// Mitsubishi GX Developer project: 11-404八軸鎖螺絲機201107140830   PLC: FX1N

PROGRAM MAIN
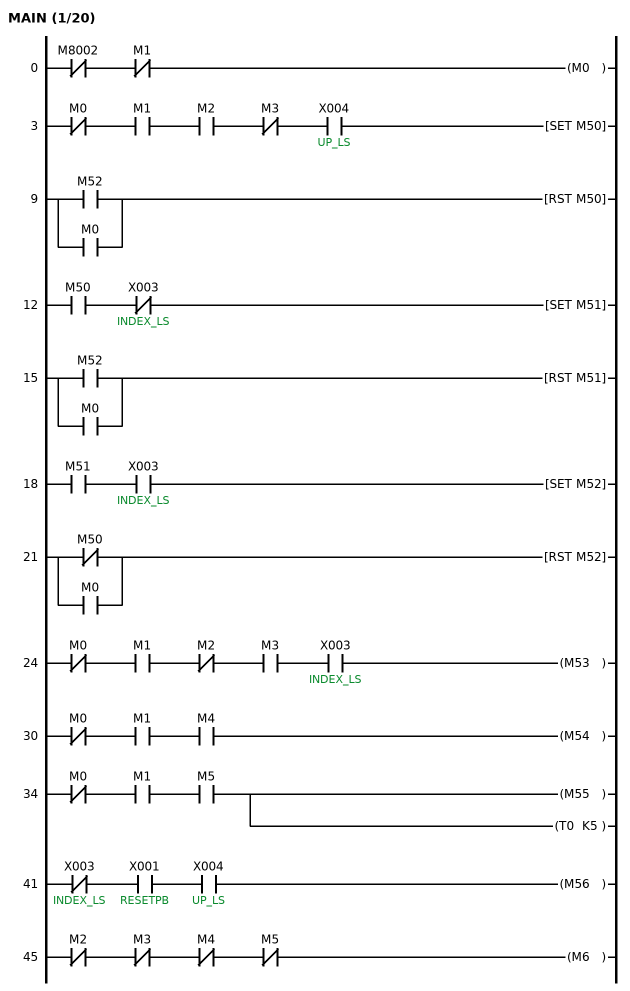
0     LDI     M8002
      ANI     M1
      OUT     M0
3     LDI     M0
      AND     M1
      AND     M2
      ANI     M3
      AND     X004  ; UP_LS
      SET     M50
9     LD      M52
      OR      M0
      RST     M50
12    LD      M50
      ANI     X003  ; INDEX_LS
      SET     M51
15    LD      M52
      OR      M0
      RST     M51
18    LD      M51
      AND     X003  ; INDEX_LS
      SET     M52
21    LDI     M50
      OR      M0
      RST     M52
24    LDI     M0
      AND     M1
      ANI     M2
      AND     M3
      AND     X003  ; INDEX_LS
      OUT     M53
30    LDI     M0
      AND     M1
      AND     M4
      OUT     M54
34    LDI     M0
      AND     M1
      AND     M5
      OUT     M55
      OUT     T0 K5
41    LDI     X003  ; INDEX_LS
      AND     X001  ; RESETPB
      AND     X004  ; UP_LS
      OUT     M56
45    LDI     M2
      ANI     M3
      ANI     M4
      ANI     M5
      OUT     M6
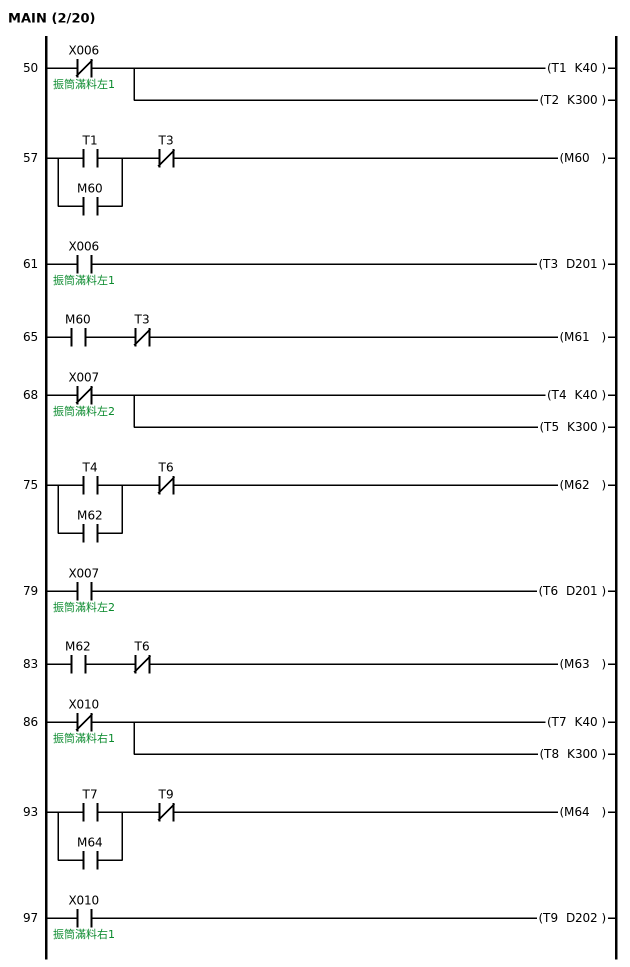
50    LDI     X006  ; 振筒滿料左1
      OUT     T1 K40
      OUT     T2 K300
57    LD      T1
      OR      M60
      ANI     T3
      OUT     M60
61    LD      X006  ; 振筒滿料左1
      OUT     T3 D201
65    LD      M60
      ANI     T3
      OUT     M61
68    LDI     X007  ; 振筒滿料左2
      OUT     T4 K40
      OUT     T5 K300
75    LD      T4
      OR      M62
      ANI     T6
      OUT     M62
79    LD      X007  ; 振筒滿料左2
      OUT     T6 D201
83    LD      M62
      ANI     T6
      OUT     M63
86    LDI     X010  ; 振筒滿料右1
      OUT     T7 K40
      OUT     T8 K300
93    LD      T7
      OR      M64
      ANI     T9
      OUT     M64
97    LD      X010  ; 振筒滿料右1
      OUT     T9 D202
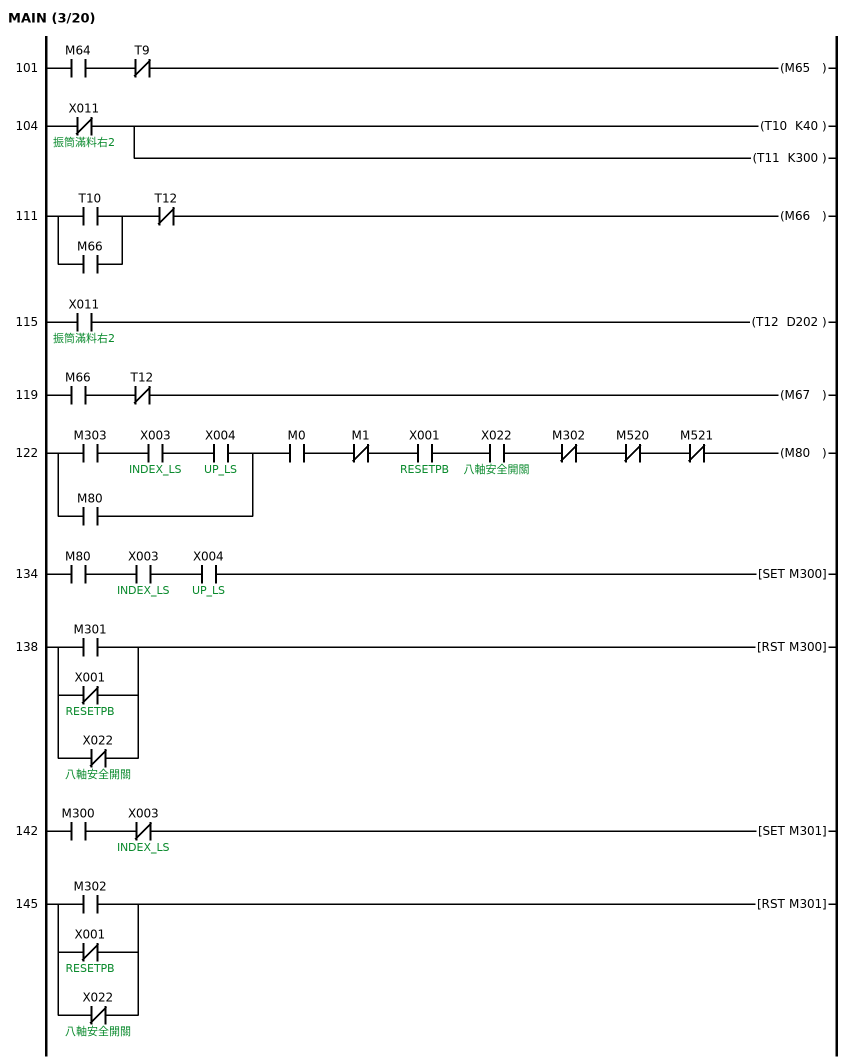
101   LD      M64
      ANI     T9
      OUT     M65
104   LDI     X011  ; 振筒滿料右2
      OUT     T10 K40
      OUT     T11 K300
111   LD      T10
      OR      M66
      ANI     T12
      OUT     M66
115   LD      X011  ; 振筒滿料右2
      OUT     T12 D202
119   LD      M66
      ANI     T12
      OUT     M67
122   LD      M303
      AND     X003  ; INDEX_LS
      AND     X004  ; UP_LS
      OR      M80
      AND     M0
      ANI     M1
      AND     X001  ; RESETPB
      AND     X022  ; 八軸安全開關
      ANI     M302
      ANI     M520
      ANI     M521
      OUT     M80
134   LD      M80
      AND     X003  ; INDEX_LS
      AND     X004  ; UP_LS
      SET     M300
138   LD      M301
      ORI     X001  ; RESETPB
      ORI     X022  ; 八軸安全開關
      RST     M300
142   LD      M300
      ANI     X003  ; INDEX_LS
      SET     M301
145   LD      M302
      ORI     X001  ; RESETPB
      ORI     X022  ; 八軸安全開關
      RST     M301
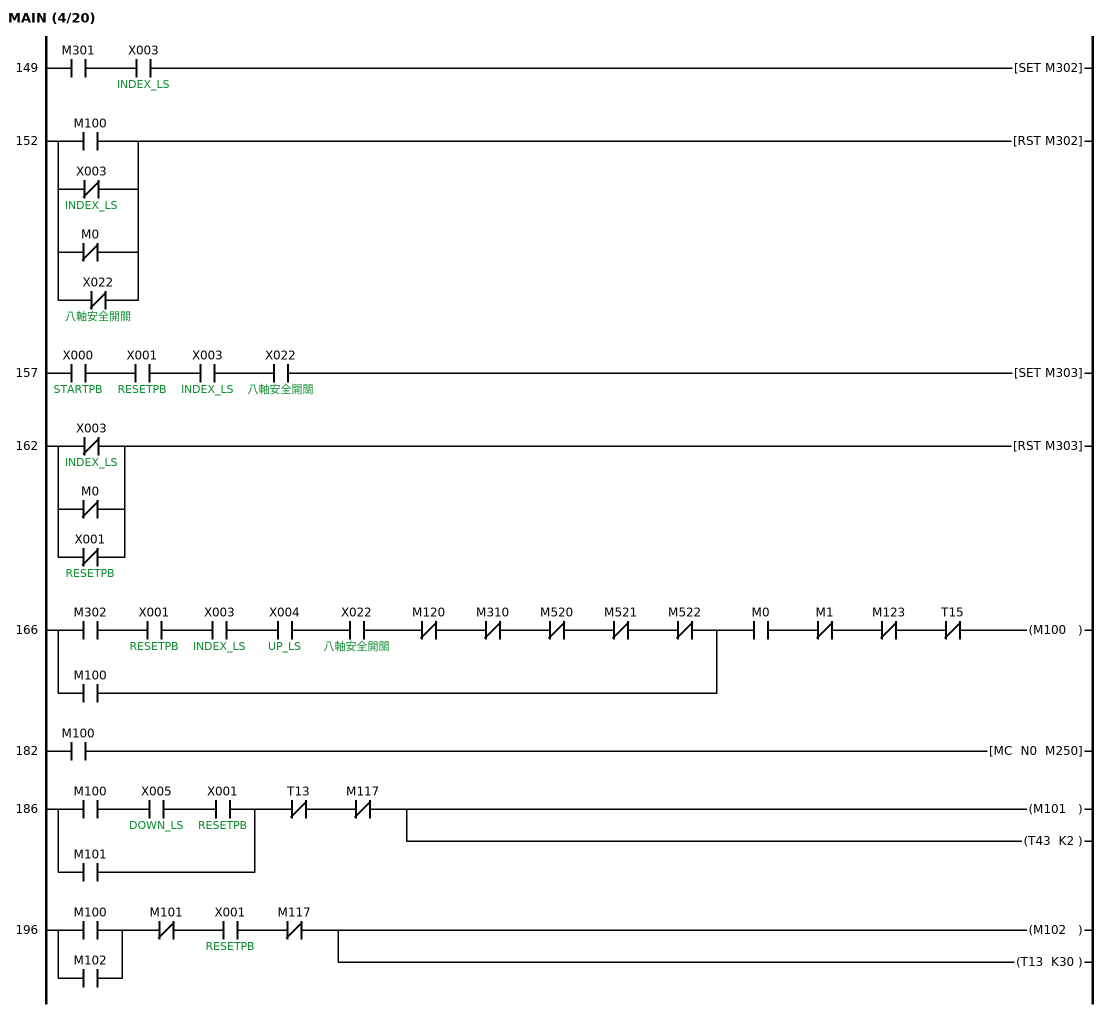
149   LD      M301
      AND     X003  ; INDEX_LS
      SET     M302
152   LD      M100
      ORI     X003  ; INDEX_LS
      ORI     M0
      ORI     X022  ; 八軸安全開關
      RST     M302
157   LD      X000  ; STARTPB
      AND     X001  ; RESETPB
      AND     X003  ; INDEX_LS
      AND     X022  ; 八軸安全開關
      SET     M303
162   LDI     X003  ; INDEX_LS
      ORI     M0
      ORI     X001  ; RESETPB
      RST     M303
166   LD      M302
      AND     X001  ; RESETPB
      AND     X003  ; INDEX_LS
      AND     X004  ; UP_LS
      AND     X022  ; 八軸安全開關
      ANI     M120
      ANI     M310
      ANI     M520
      ANI     M521
      ANI     M522
      OR      M100
      AND     M0
      ANI     M1
      ANI     M123
      ANI     T15
      OUT     M100
182   LD      M100
      MC      N0 M250
186   LD      M100
      AND     X005  ; DOWN_LS
      AND     X001  ; RESETPB
      OR      M101
      ANI     T13
      ANI     M117
      OUT     M101
      OUT     T43 K2
196   LD      M100
      OR      M102
      ANI     M101
      AND     X001  ; RESETPB
      ANI     M117
      OUT     M102
      OUT     T13 K30
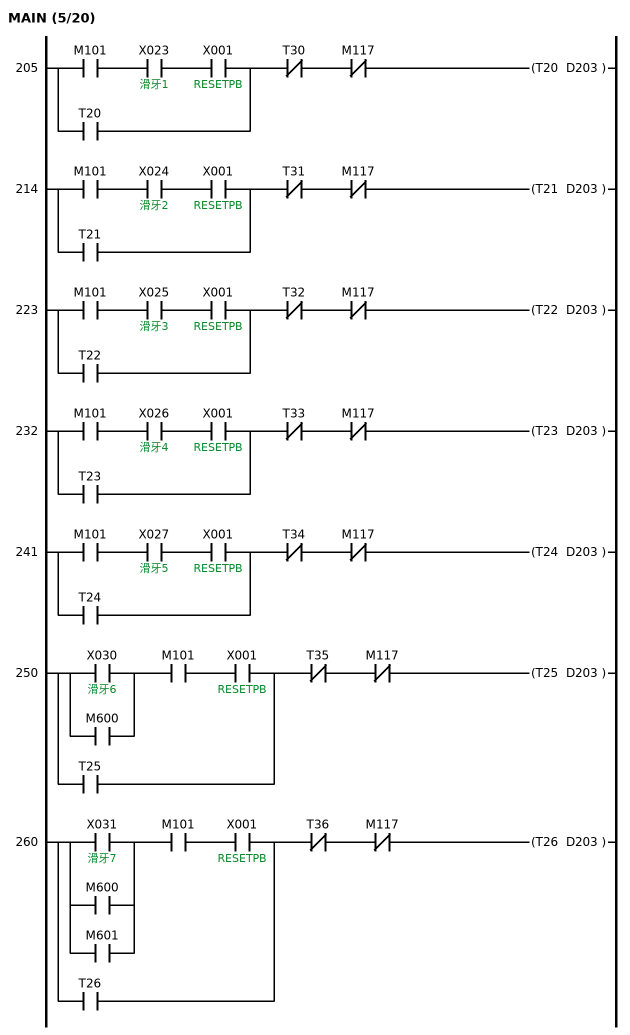
205   LD      M101
      AND     X023  ; 滑牙1
      AND     X001  ; RESETPB
      OR      T20
      ANI     T30
      ANI     M117
      OUT     T20 D203
214   LD      M101
      AND     X024  ; 滑牙2
      AND     X001  ; RESETPB
      OR      T21
      ANI     T31
      ANI     M117
      OUT     T21 D203
223   LD      M101
      AND     X025  ; 滑牙3
      AND     X001  ; RESETPB
      OR      T22
      ANI     T32
      ANI     M117
      OUT     T22 D203
232   LD      M101
      AND     X026  ; 滑牙4
      AND     X001  ; RESETPB
      OR      T23
      ANI     T33
      ANI     M117
      OUT     T23 D203
241   LD      M101
      AND     X027  ; 滑牙5
      AND     X001  ; RESETPB
      OR      T24
      ANI     T34
      ANI     M117
      OUT     T24 D203
250   LD      X030  ; 滑牙6
      OR      M600
      AND     M101
      AND     X001  ; RESETPB
      OR      T25
      ANI     T35
      ANI     M117
      OUT     T25 D203
260   LD      X031  ; 滑牙7
      OR      M600
      OR      M601
      AND     M101
      AND     X001  ; RESETPB
      OR      T26
      ANI     T36
      ANI     M117
      OUT     T26 D203
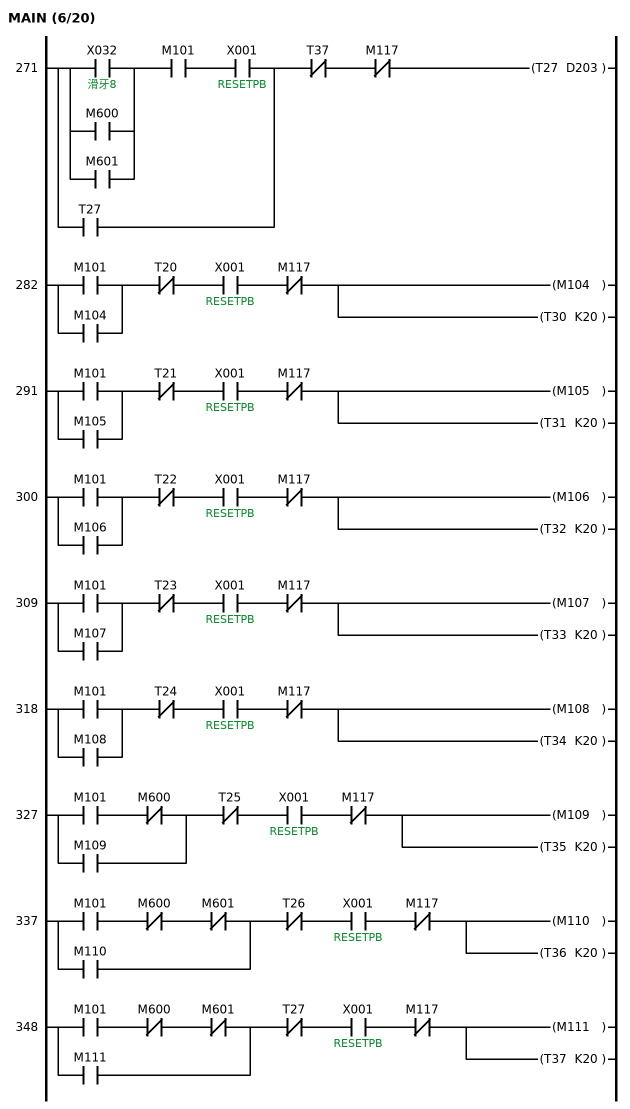
271   LD      X032  ; 滑牙8
      OR      M600
      OR      M601
      AND     M101
      AND     X001  ; RESETPB
      OR      T27
      ANI     T37
      ANI     M117
      OUT     T27 D203
282   LD      M101
      OR      M104
      ANI     T20
      AND     X001  ; RESETPB
      ANI     M117
      OUT     M104
      OUT     T30 K20
291   LD      M101
      OR      M105
      ANI     T21
      AND     X001  ; RESETPB
      ANI     M117
      OUT     M105
      OUT     T31 K20
300   LD      M101
      OR      M106
      ANI     T22
      AND     X001  ; RESETPB
      ANI     M117
      OUT     M106
      OUT     T32 K20
309   LD      M101
      OR      M107
      ANI     T23
      AND     X001  ; RESETPB
      ANI     M117
      OUT     M107
      OUT     T33 K20
318   LD      M101
      OR      M108
      ANI     T24
      AND     X001  ; RESETPB
      ANI     M117
      OUT     M108
      OUT     T34 K20
327   LD      M101
      ANI     M600
      OR      M109
      ANI     T25
      AND     X001  ; RESETPB
      ANI     M117
      OUT     M109
      OUT     T35 K20
337   LD      M101
      ANI     M600
      ANI     M601
      OR      M110
      ANI     T26
      AND     X001  ; RESETPB
      ANI     M117
      OUT     M110
      OUT     T36 K20
348   LD      M101
      ANI     M600
      ANI     M601
      OR      M111
      ANI     T27
      AND     X001  ; RESETPB
      ANI     M117
      OUT     M111
      OUT     T37 K20
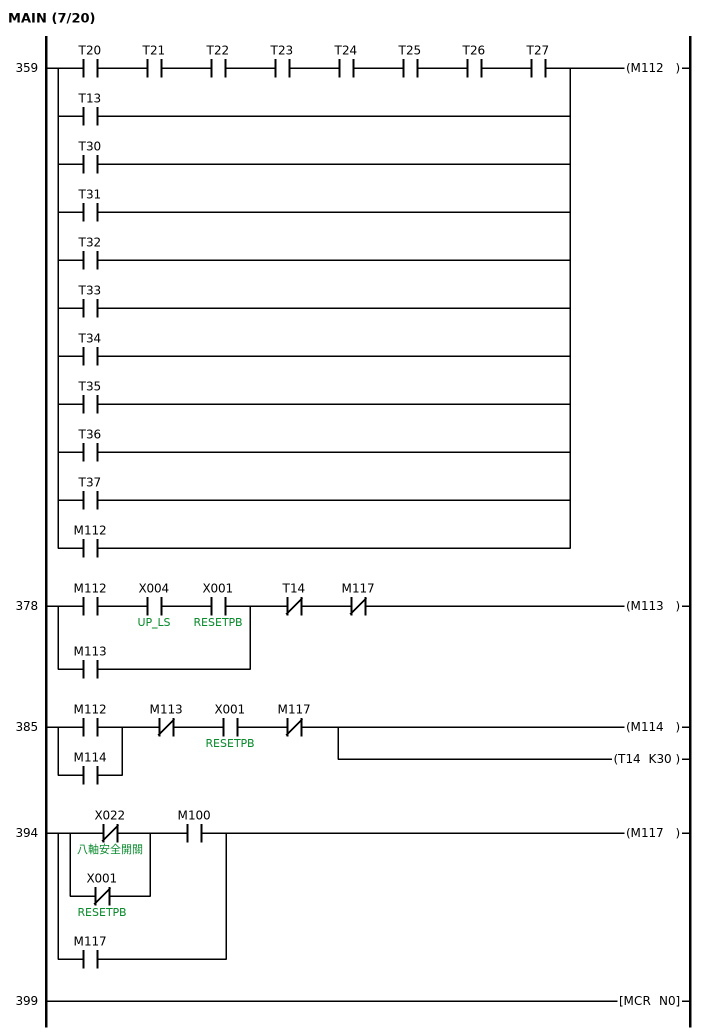
359   LD      T20
      AND     T21
      AND     T22
      AND     T23
      AND     T24
      AND     T25
      AND     T26
      AND     T27
      OR      T13
      OR      T30
      OR      T31
      OR      T32
      OR      T33
      OR      T34
      OR      T35
      OR      T36
      OR      T37
      OR      M112
      OUT     M112
378   LD      M112
      AND     X004  ; UP_LS
      AND     X001  ; RESETPB
      OR      M113
      ANI     T14
      ANI     M117
      OUT     M113
385   LD      M112
      OR      M114
      ANI     M113
      AND     X001  ; RESETPB
      ANI     M117
      OUT     M114
      OUT     T14 K30
394   LDI     X022  ; 八軸安全開關
      ORI     X001  ; RESETPB
      AND     M100
      OR      M117
      OUT     M117
399   MCR     N0
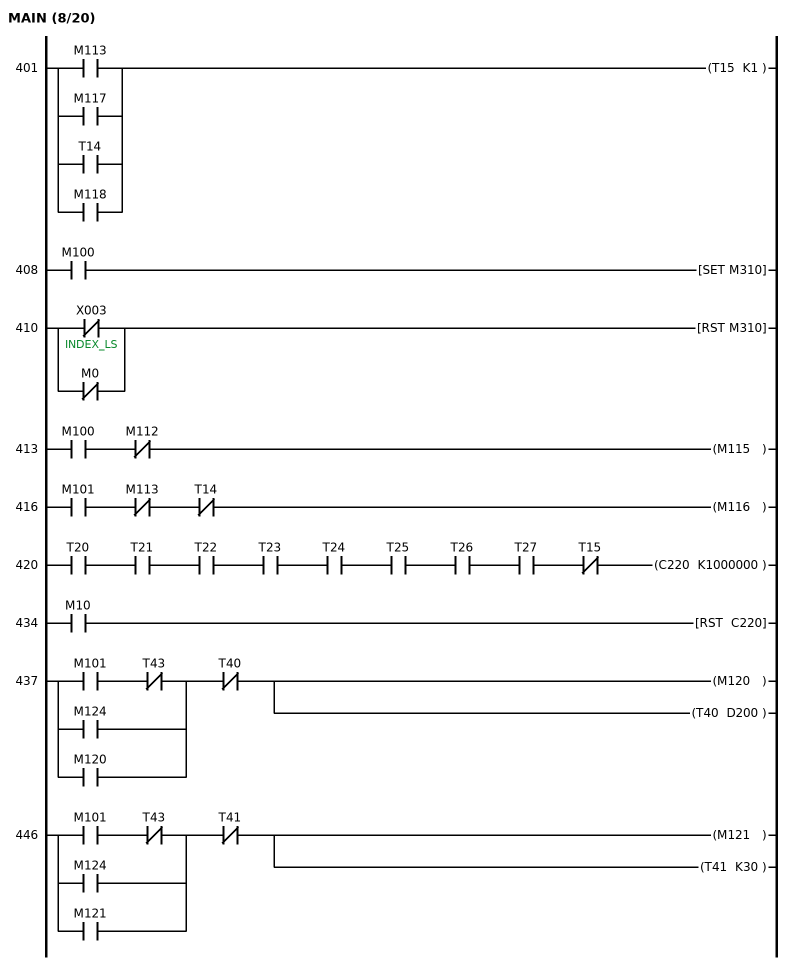
401   LD      M113
      OR      M117
      OR      T14
      OR      M118
      OUT     T15 K1
408   LD      M100
      SET     M310
410   LDI     X003  ; INDEX_LS
      ORI     M0
      RST     M310
413   LD      M100
      ANI     M112
      OUT     M115
416   LD      M101
      ANI     M113
      ANI     T14
      OUT     M116
420   LD      T20
      AND     T21
      AND     T22
      AND     T23
      AND     T24
      AND     T25
      AND     T26
      AND     T27
      ANI     T15
      OUT     C220 K1000000
434   LD      M10
      RST     C220
437   LD      M101
      ANI     T43
      OR      M124
      OR      M120
      ANI     T40
      OUT     M120
      OUT     T40 D200
446   LD      M101
      ANI     T43
      OR      M124
      OR      M121
      ANI     T41
      OUT     M121
      OUT     T41 K30
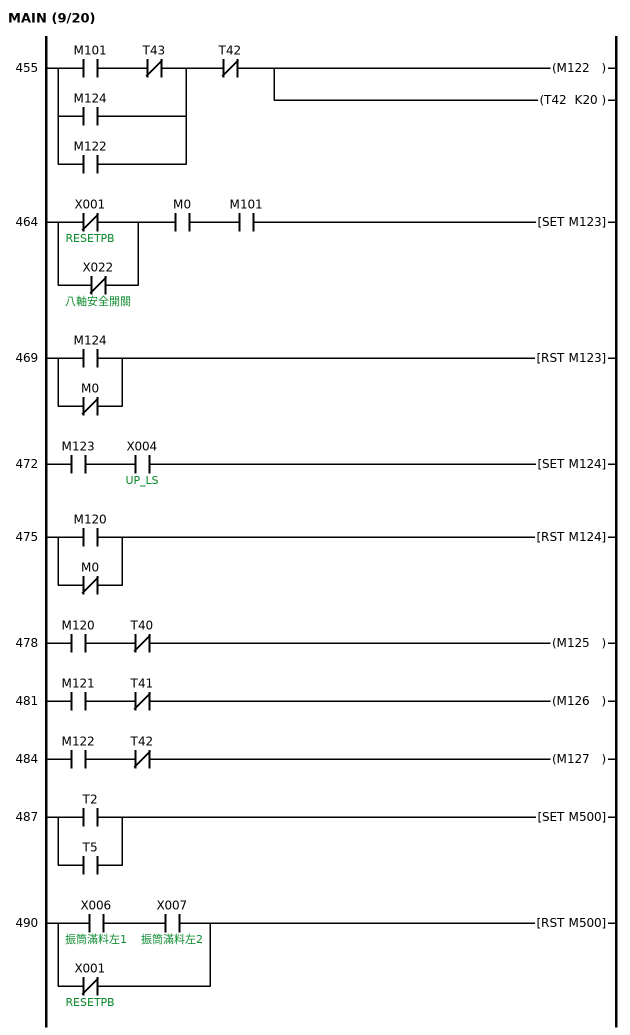
455   LD      M101
      ANI     T43
      OR      M124
      OR      M122
      ANI     T42
      OUT     M122
      OUT     T42 K20
464   LDI     X001  ; RESETPB
      ORI     X022  ; 八軸安全開關
      AND     M0
      AND     M101
      SET     M123
469   LD      M124
      ORI     M0
      RST     M123
472   LD      M123
      AND     X004  ; UP_LS
      SET     M124
475   LD      M120
      ORI     M0
      RST     M124
478   LD      M120
      ANI     T40
      OUT     M125
481   LD      M121
      ANI     T41
      OUT     M126
484   LD      M122
      ANI     T42
      OUT     M127
487   LD      T2
      OR      T5
      SET     M500
490   LD      X006  ; 振筒滿料左1
      AND     X007  ; 振筒滿料左2
      ORI     X001  ; RESETPB
      RST     M500
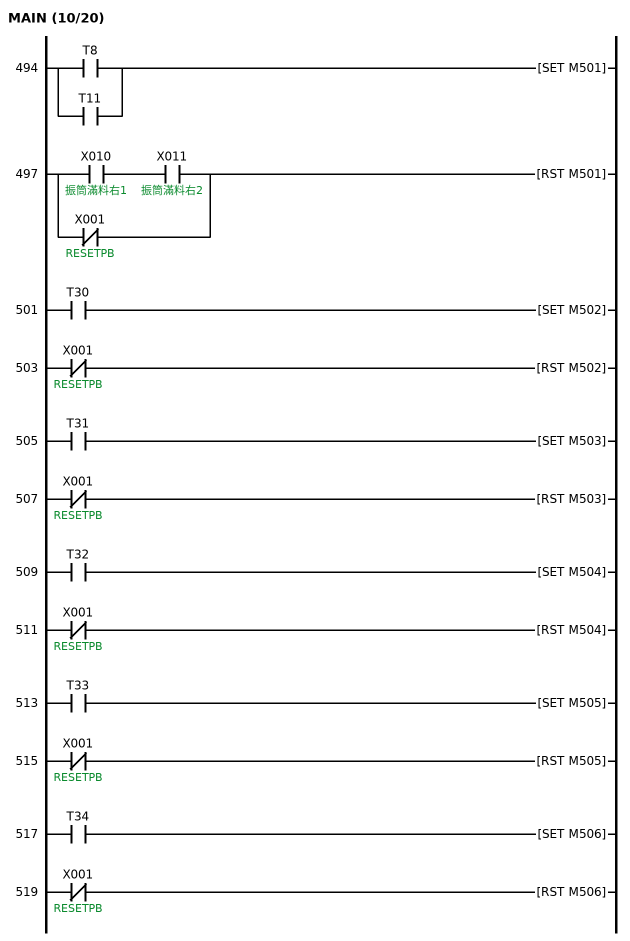
494   LD      T8
      OR      T11
      SET     M501
497   LD      X010  ; 振筒滿料右1
      AND     X011  ; 振筒滿料右2
      ORI     X001  ; RESETPB
      RST     M501
501   LD      T30
      SET     M502
503   LDI     X001  ; RESETPB
      RST     M502
505   LD      T31
      SET     M503
507   LDI     X001  ; RESETPB
      RST     M503
509   LD      T32
      SET     M504
511   LDI     X001  ; RESETPB
      RST     M504
513   LD      T33
      SET     M505
515   LDI     X001  ; RESETPB
      RST     M505
517   LD      T34
      SET     M506
519   LDI     X001  ; RESETPB
      RST     M506
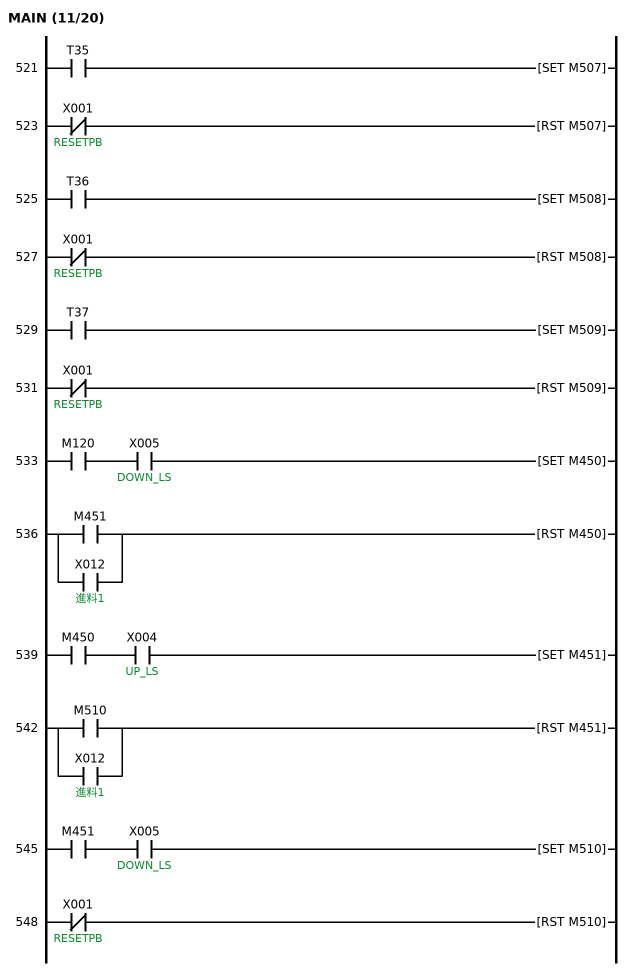
521   LD      T35
      SET     M507
523   LDI     X001  ; RESETPB
      RST     M507
525   LD      T36
      SET     M508
527   LDI     X001  ; RESETPB
      RST     M508
529   LD      T37
      SET     M509
531   LDI     X001  ; RESETPB
      RST     M509
533   LD      M120
      AND     X005  ; DOWN_LS
      SET     M450
536   LD      M451
      OR      X012  ; 進料1
      RST     M450
539   LD      M450
      AND     X004  ; UP_LS
      SET     M451
542   LD      M510
      OR      X012  ; 進料1
      RST     M451
545   LD      M451
      AND     X005  ; DOWN_LS
      SET     M510
548   LDI     X001  ; RESETPB
      RST     M510
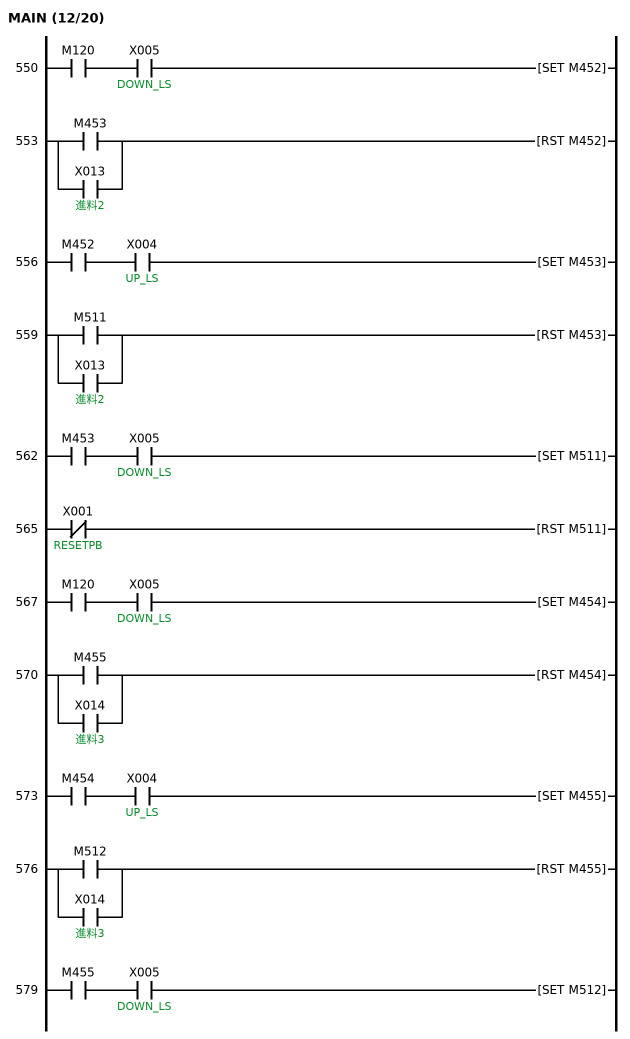
550   LD      M120
      AND     X005  ; DOWN_LS
      SET     M452
553   LD      M453
      OR      X013  ; 進料2
      RST     M452
556   LD      M452
      AND     X004  ; UP_LS
      SET     M453
559   LD      M511
      OR      X013  ; 進料2
      RST     M453
562   LD      M453
      AND     X005  ; DOWN_LS
      SET     M511
565   LDI     X001  ; RESETPB
      RST     M511
567   LD      M120
      AND     X005  ; DOWN_LS
      SET     M454
570   LD      M455
      OR      X014  ; 進料3
      RST     M454
573   LD      M454
      AND     X004  ; UP_LS
      SET     M455
576   LD      M512
      OR      X014  ; 進料3
      RST     M455
579   LD      M455
      AND     X005  ; DOWN_LS
      SET     M512
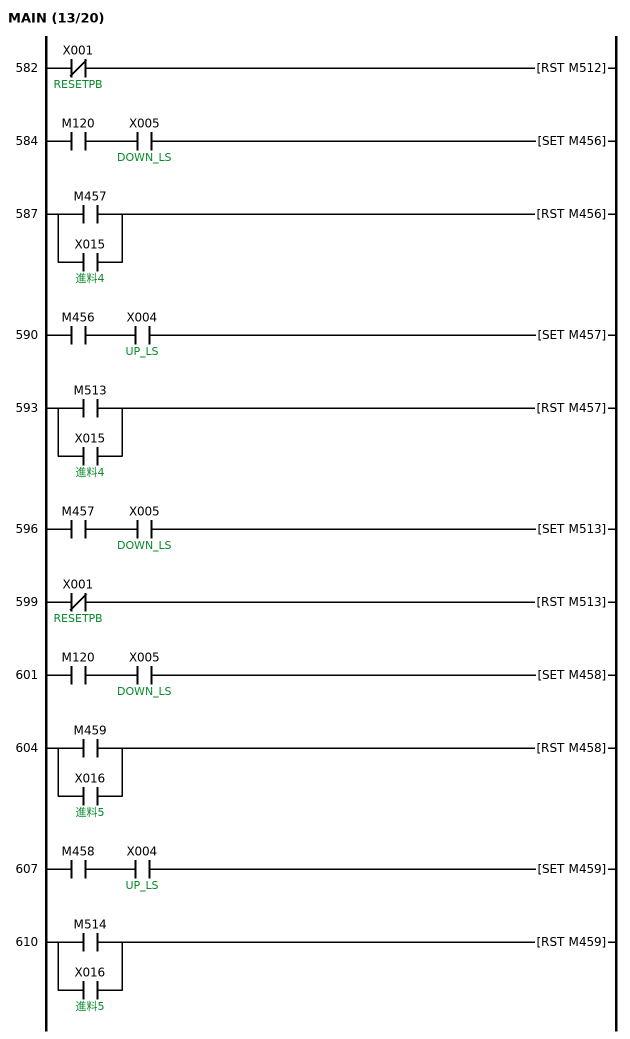
582   LDI     X001  ; RESETPB
      RST     M512
584   LD      M120
      AND     X005  ; DOWN_LS
      SET     M456
587   LD      M457
      OR      X015  ; 進料4
      RST     M456
590   LD      M456
      AND     X004  ; UP_LS
      SET     M457
593   LD      M513
      OR      X015  ; 進料4
      RST     M457
596   LD      M457
      AND     X005  ; DOWN_LS
      SET     M513
599   LDI     X001  ; RESETPB
      RST     M513
601   LD      M120
      AND     X005  ; DOWN_LS
      SET     M458
604   LD      M459
      OR      X016  ; 進料5
      RST     M458
607   LD      M458
      AND     X004  ; UP_LS
      SET     M459
610   LD      M514
      OR      X016  ; 進料5
      RST     M459
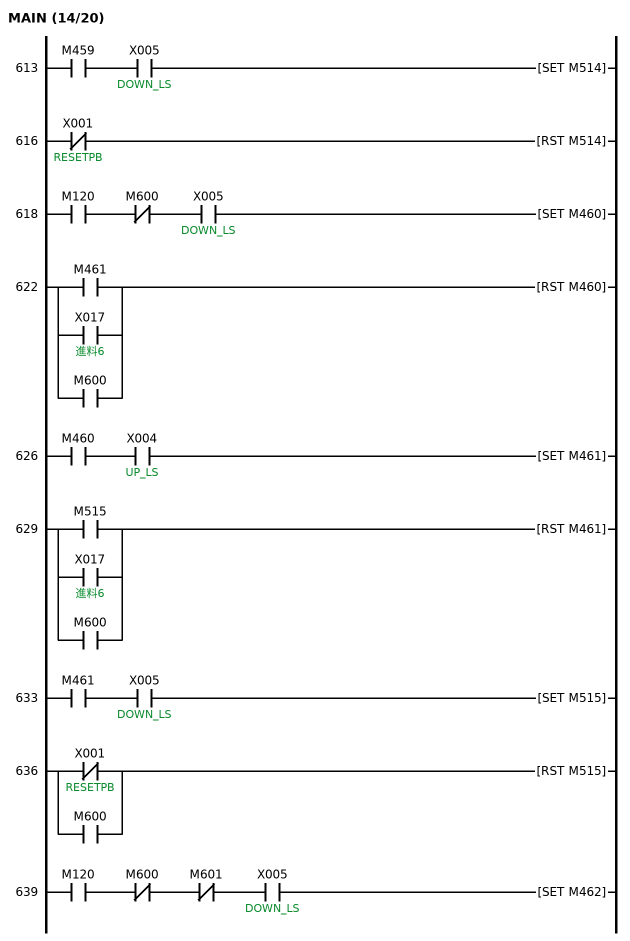
613   LD      M459
      AND     X005  ; DOWN_LS
      SET     M514
616   LDI     X001  ; RESETPB
      RST     M514
618   LD      M120
      ANI     M600
      AND     X005  ; DOWN_LS
      SET     M460
622   LD      M461
      OR      X017  ; 進料6
      OR      M600
      RST     M460
626   LD      M460
      AND     X004  ; UP_LS
      SET     M461
629   LD      M515
      OR      X017  ; 進料6
      OR      M600
      RST     M461
633   LD      M461
      AND     X005  ; DOWN_LS
      SET     M515
636   LDI     X001  ; RESETPB
      OR      M600
      RST     M515
639   LD      M120
      ANI     M600
      ANI     M601
      AND     X005  ; DOWN_LS
      SET     M462
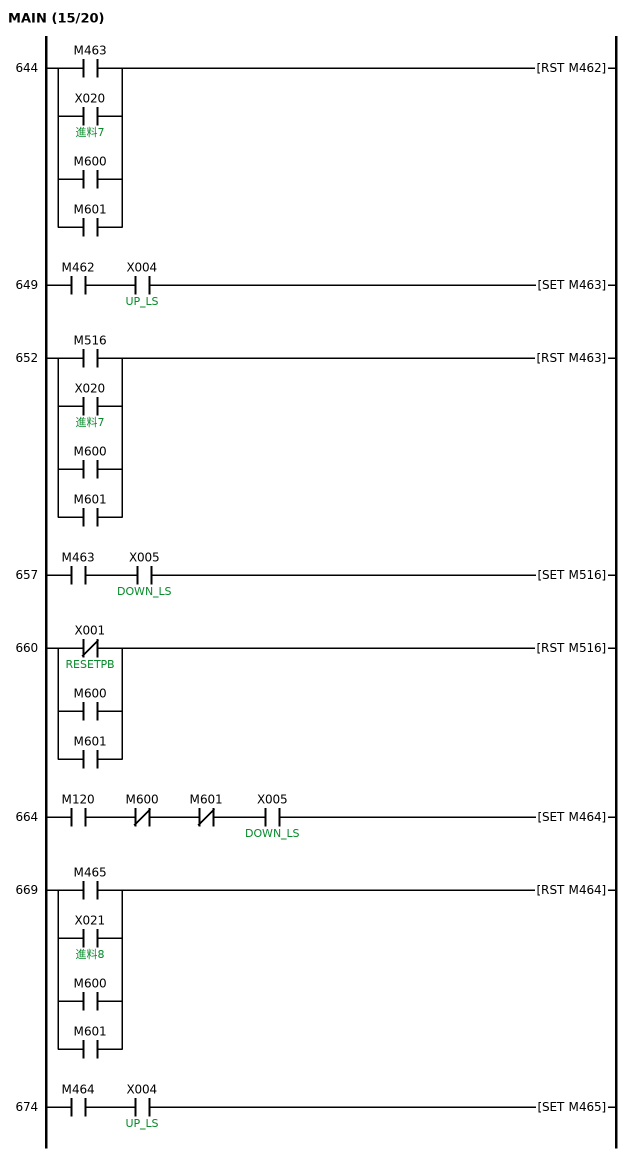
644   LD      M463
      OR      X020  ; 進料7
      OR      M600
      OR      M601
      RST     M462
649   LD      M462
      AND     X004  ; UP_LS
      SET     M463
652   LD      M516
      OR      X020  ; 進料7
      OR      M600
      OR      M601
      RST     M463
657   LD      M463
      AND     X005  ; DOWN_LS
      SET     M516
660   LDI     X001  ; RESETPB
      OR      M600
      OR      M601
      RST     M516
664   LD      M120
      ANI     M600
      ANI     M601
      AND     X005  ; DOWN_LS
      SET     M464
669   LD      M465
      OR      X021  ; 進料8
      OR      M600
      OR      M601
      RST     M464
674   LD      M464
      AND     X004  ; UP_LS
      SET     M465
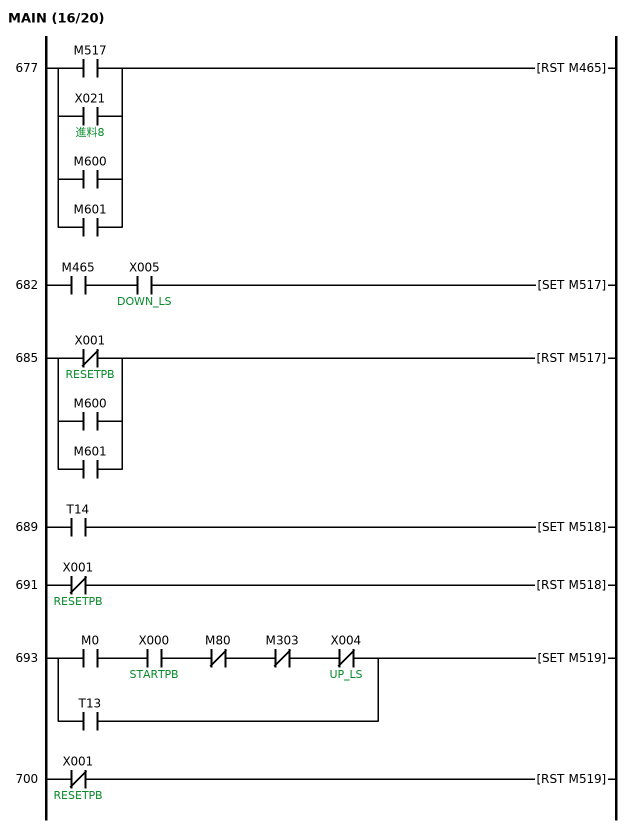
677   LD      M517
      OR      X021  ; 進料8
      OR      M600
      OR      M601
      RST     M465
682   LD      M465
      AND     X005  ; DOWN_LS
      SET     M517
685   LDI     X001  ; RESETPB
      OR      M600
      OR      M601
      RST     M517
689   LD      T14
      SET     M518
691   LDI     X001  ; RESETPB
      RST     M518
693   LD      M0
      AND     X000  ; STARTPB
      ANI     M80
      ANI     M303
      ANI     X004  ; UP_LS
      OR      T13
      SET     M519
700   LDI     X001  ; RESETPB
      RST     M519
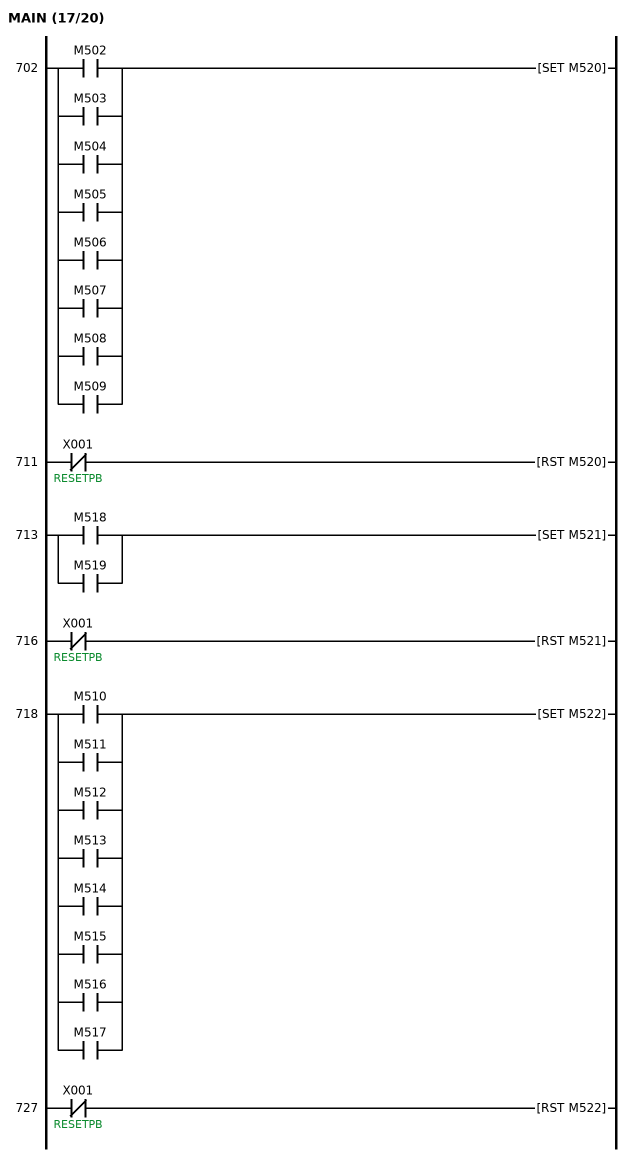
702   LD      M502
      OR      M503
      OR      M504
      OR      M505
      OR      M506
      OR      M507
      OR      M508
      OR      M509
      SET     M520
711   LDI     X001  ; RESETPB
      RST     M520
713   LD      M518
      OR      M519
      SET     M521
716   LDI     X001  ; RESETPB
      RST     M521
718   LD      M510
      OR      M511
      OR      M512
      OR      M513
      OR      M514
      OR      M515
      OR      M516
      OR      M517
      SET     M522
727   LDI     X001  ; RESETPB
      RST     M522
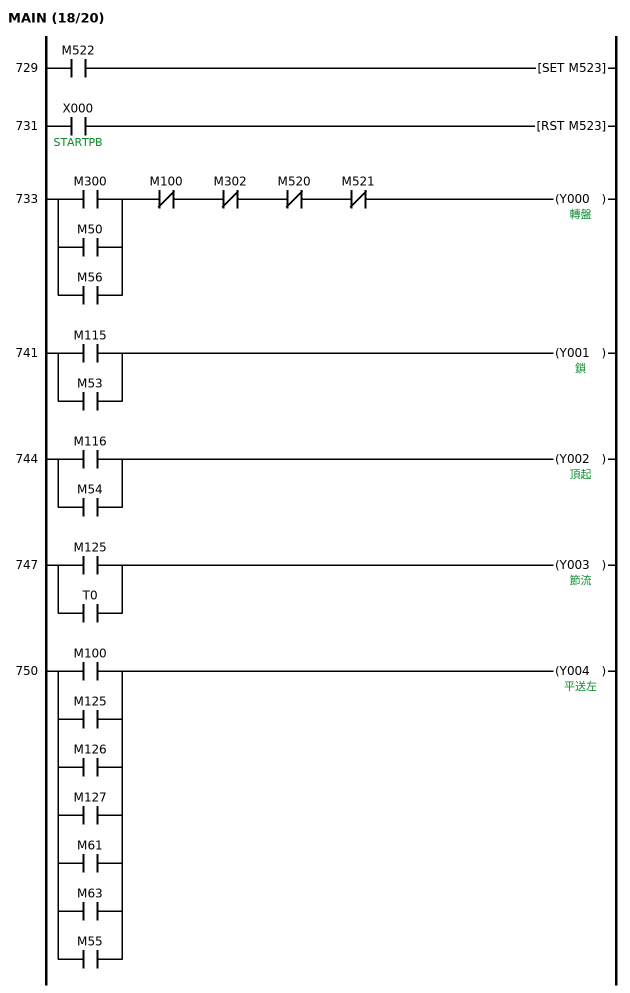
729   LD      M522
      SET     M523
731   LD      X000  ; STARTPB
      RST     M523
733   LD      M300
      OR      M50
      OR      M56
      ANI     M100
      ANI     M302
      ANI     M520
      ANI     M521
      OUT     Y000  ; 轉盤
741   LD      M115
      OR      M53
      OUT     Y001  ; 鎖
744   LD      M116
      OR      M54
      OUT     Y002  ; 頂起
747   LD      M125
      OR      T0
      OUT     Y003  ; 節流
750   LD      M100
      OR      M125
      OR      M126
      OR      M127
      OR      M61
      OR      M63
      OR      M55
      OUT     Y004  ; 平送左
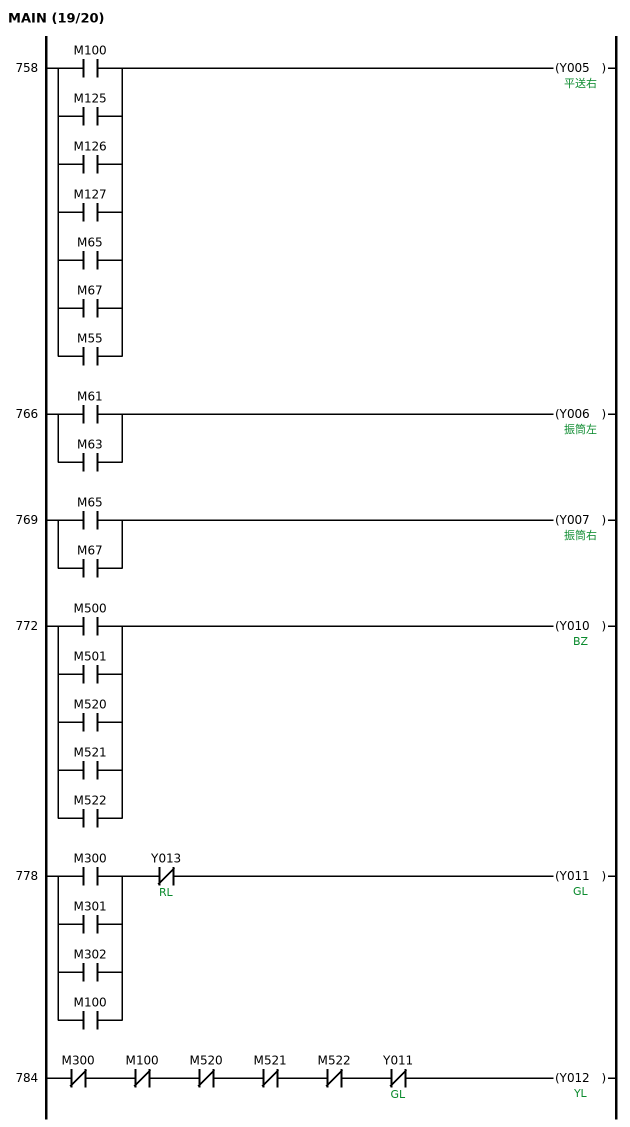
758   LD      M100
      OR      M125
      OR      M126
      OR      M127
      OR      M65
      OR      M67
      OR      M55
      OUT     Y005  ; 平送右
766   LD      M61
      OR      M63
      OUT     Y006  ; 振筒左
769   LD      M65
      OR      M67
      OUT     Y007  ; 振筒右
772   LD      M500
      OR      M501
      OR      M520
      OR      M521
      OR      M522
      OUT     Y010  ; BZ
778   LD      M300
      OR      M301
      OR      M302
      OR      M100
      ANI     Y013  ; RL
      OUT     Y011  ; GL
784   LDI     M300
      ANI     M100
      ANI     M520
      ANI     M521
      ANI     M522
      ANI     Y011  ; GL
      OUT     Y012  ; YL
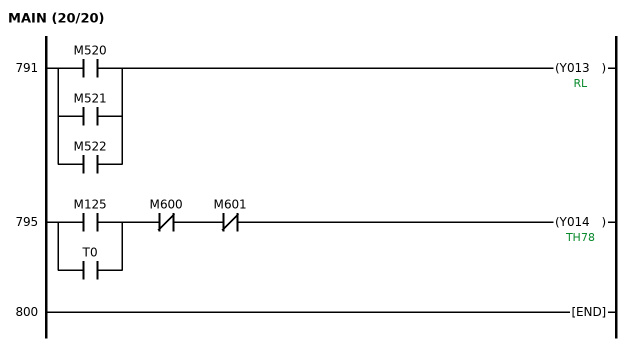
791   LD      M520
      OR      M521
      OR      M522
      OUT     Y013  ; RL
795   LD      M125
      OR      T0
      ANI     M600
      ANI     M601
      OUT     Y014  ; TH78
800   END
END_PROGRAM

// device comments not shown above
Y015  ; TH12
Y016  ; TH34
Y017  ; TH56
